DATA_BLOCK "DB_Parm"
{ S7_Optimized_Access := 'TRUE' }
VERSION : 0.1
NON_RETAIN
   VAR

      StationNo : Int := 2;
      tClamp : Time := T#500MS;
      tTableMove : Time := T#1S;
      tHeadDown : Time := T#1S;
      tAlarmDelay : Time := T#2S;
   END_VAR
BEGIN
END_DATA_BLOCK
